FUNCTION F_TrueBitsCounter : UINT
VAR_INPUT
	pArray			: POINTER TO ARRAY[0..255] OF BOOL;
	arrBitSize		: UINT; 
END_VAR
	
VAR
	i				: UINT;
END_VAR



FOR i:=0 TO arrBitSize-1 DO
	IF pArray^[i] THEN
		F_TrueBitsCounter	:= F_TrueBitsCounter + 1;
	END_IF
END_FOR

END_FUNCTION

(* stored: Version 1.1.0.1, ProductVersion 3.1.4024.12
   POU F_TrueBitsCounter: Id {b9c43333-8d95-4a59-b7a9-8460dce32864}, SpecialFunc None *)
